// SIMATIC S7-200 project (STEP 7-Micro/WIN), CPU 221 REL 01.10

SYMBOL_TABLE USUARIO1
S1               I0.0     // Sensor magnético que detecta pistón 1 contraído (NA)
S2               I0.1     // Sensor magnético que detecta pistón 1 expandido (NA)
S3               I0.2     // Switch final de carrera que detecta cuando cae una bolsa (NA)
S4               I0.3     // Sensor fotoeléctrico que detecta una bolsa en la banda (NA)
S5               I0.4     // Sensor fotoeléctrico que sirve para contar las bolsas (NA)
S6               I0.5     // Sensor magnético que detecta pistón 1 contraído (NA)
S7               I0.6     // Sensor magnético que detecta pistón 1 expandido (NA)
S8               I0.7     // Sensor fotoeléctrico que detecta una bolsa en la banda (NA)
S9               I1.0     // Switch final de carrera que detecta puerta cerrada (NA)
S10              I1.1     // Switch final de carrera que detecta puerta abierta (NA)
DAR_BOLSA        Q0.0     // Activar el alimentador de bolsas
SACAR_PISTON_1   Q0.1     // Expandir el pistón 1
METER_PISTON_1   Q0.2     // Contraer el pistón 1
BANDAS_CONTAJE   Q0.3     // Encender bandas que llevan las bolsas al contador
SACAR_PISTON_2   Q0.4     // Expandir el pistón 2
METER_PISTON_2   Q0.5     // Contraer el pistón 2
LED              Q0.6     // Señalización que indica cuando han pasado 3 bolsas
BANDAS_EMPAQUE   Q0.7     // Encender bandas que llevan las bolsas a la puerta
ABRIR_PUERTA     Q1.0     // Abrir puerta
CERRAR_PUERTA    Q1.1     // Cerrar puerta
END_SYMBOL_TABLE

ORGANIZATION_BLOCK PRINCIPAL:OB1
TITLE=COMENTARIOS DEL PROGRAMA
BEGIN
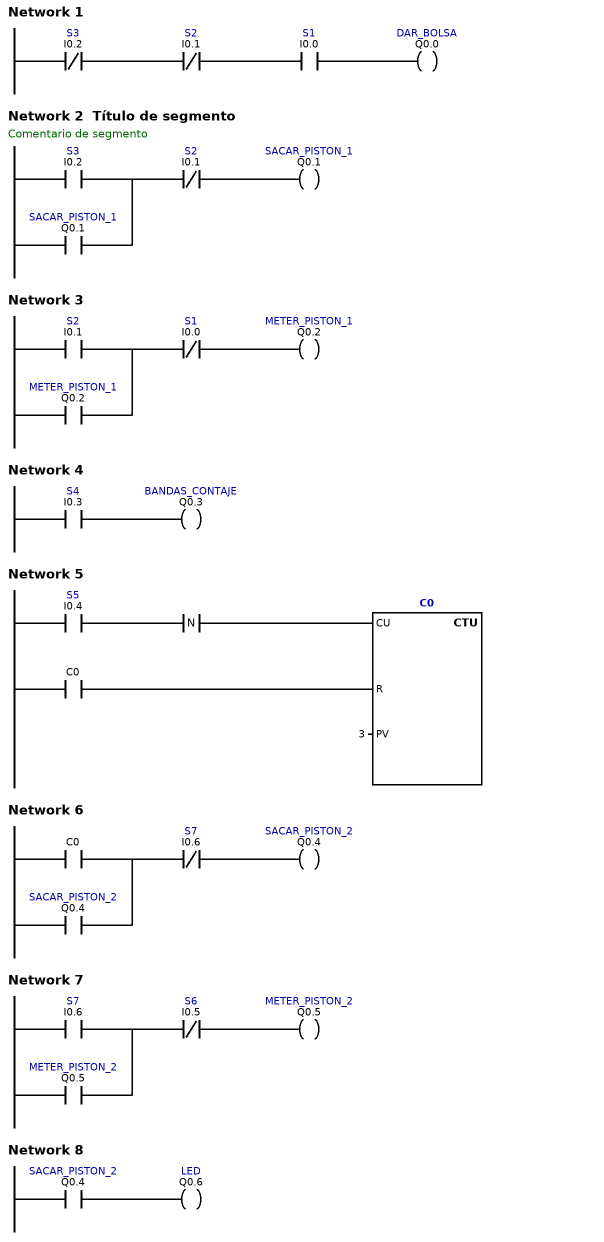
Network 1
LDN    S3:I0.2
AN     S2:I0.1
A      S1:I0.0
=      DAR_BOLSA:Q0.0
Network 2 // Título de segmento
// Comentario de segmento
LD     S3:I0.2
O      SACAR_PISTON_1:Q0.1
AN     S2:I0.1
=      SACAR_PISTON_1:Q0.1
Network 3
LD     S2:I0.1
O      METER_PISTON_1:Q0.2
AN     S1:I0.0
=      METER_PISTON_1:Q0.2
Network 4
LD     S4:I0.3
=      BANDAS_CONTAJE:Q0.3
Network 5
LD     S5:I0.4
ED
LD     C0
CTU    C0, 3
Network 6
LD     C0
O      SACAR_PISTON_2:Q0.4
AN     S7:I0.6
=      SACAR_PISTON_2:Q0.4
Network 7
LD     S7:I0.6
O      METER_PISTON_2:Q0.5
AN     S6:I0.5
=      METER_PISTON_2:Q0.5
Network 8
LD     SACAR_PISTON_2:Q0.4
=      LED:Q0.6
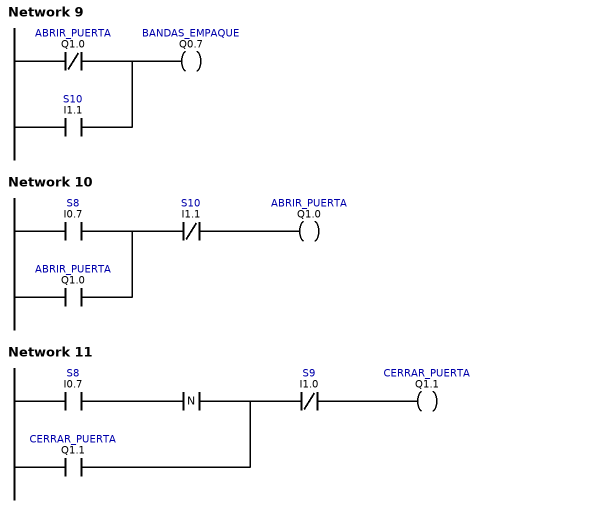
Network 9
LDN    ABRIR_PUERTA:Q1.0
O      S10:I1.1
=      BANDAS_EMPAQUE:Q0.7
Network 10
LD     S8:I0.7
O      ABRIR_PUERTA:Q1.0
AN     S10:I1.1
=      ABRIR_PUERTA:Q1.0
Network 11
LD     S8:I0.7
ED
O      CERRAR_PUERTA:Q1.1
AN     S9:I1.0
=      CERRAR_PUERTA:Q1.1
END_ORGANIZATION_BLOCK
